// TIA Portal V19 export
DATA_BLOCK "Robot_Modbus_DB"   // DB1
// stored: InstanceOfName Robot_Modbus, InstanceOfType FB
"Robot_Modbus"
   // VAR_INPUT
   //    Proces_Item : Bool;
   //    Place_Item_Conveyor : Bool;
   //    Place_Item_Storage : Bool;
   //    Scrap_Item : Bool;
   //    Speed_Transport : Int;
   //    Speed_Grinding : Int;
   //    Grinding_Coordinates : Bool;
   //    HMI_String : String;
   // END_VAR
   // VAR_OUTPUT
   //    Working : Bool;
   //    Done : Bool;
   //    Error : Bool;
   //    Reached_Coordinates : Bool;
   // END_VAR
   // VAR
   //    DISCONNECT : Bool;
   //    Address : TCON_IP_v4;
   //    Receive_Data : Int;
   //    Send_Data : Array[0..63] of Bool;
   //    Send_Coordinates : Array[0..2] of Int;
   //    Letter_A : Array[0..20] of "XYZ_Coordinates";
   //    Letter_Steps { S7_SetPoint := 'True'} : Int;
   //    Rising_edge : Bool;
   //    String_To_Letter_Array : Array[0..16] of Char;
   //    String_Length : Int;
   //    Currently_Processing : Int;
   //    Send_Letter_A : Bool;
   //    Send_Letter_B : Bool;
   //    Send_Letter_C : Bool;
   //    MB_Client_Mode : Int;
   //    MB_Client_Modbus_Address : Int;
   //    For_Loop_Counter : Int;
   // END_VAR
BEGIN
END_DATA_BLOCK
